ABB RobotStudio station: ESTACION_DEF_ROBOT.rsstn

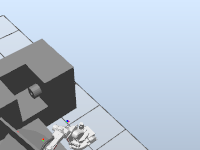
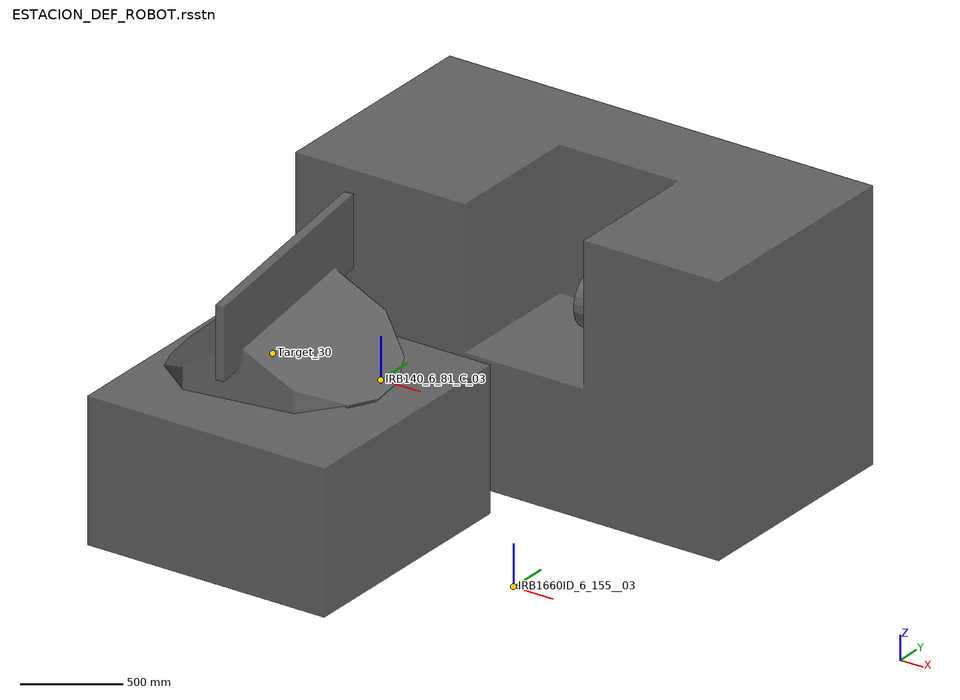
[picture v1: parts stored in the station drawn from their meshes, with robot base, taught points and paths (robot models come from the ABB library and are not in the file)]
Station ESTACION_DEF_ROBOT (saved by RobotStudio 21.2.9526.0)
Controller Controlador6, task T_ROB1: task frame (RAPID world) sits at (1882.6, -1569.1, 39.06) mm, rotated rx 0 ry 0 rz 180 deg in the station
Controller Controlador5
  mechanical unit ROB_1: IRB140_6_81_C_03, 6 joints, base frame (0, 0, 0) mm
Controller Controlador6
  mechanical unit ROB_1: IRB1660ID_6_155__03, 6 joints, base frame (0, 0, 0) mm
Layout (positions relative to the parent item):
  - IRB140_6_81_C_03 [mechanism, from Robots\IRB140_6_81_C_G_03.rslib] at (0, 0, 0) mm; joint values [0, -0.1562, 0.2279, 0, 0.4519, 0] (rad or m)
  - Conjunto_para_piezas_2 [part] at (0, 0, 452.24) mm, rotated rx 90 ry 0 rz 0 deg, size 1400 x 1500 x 1400 mm
  - IRB1660ID_6_155__03 [mechanism, from Robots\IRB1660ID_6_155__03.rslib] at (1882.6, -1569.1, 39.06) mm, rotated rx 0 ry 0 rz 180 deg; joint values [0, 0, 0, 0, 0.5236, 0] (rad or m)
  - Torno [part] at (2480.52, 608.66, 1496.19) mm, rotated rx 0 ry 0 rz 180 deg, size 2500 x 1300 x 1500 mm
  - MyTool_2 [mechanism, from Training Objects\myTool.rslib] at (726.72, -1949.96, 1124.78) mm, rotated rx 180 ry 0 rz 0 deg
Attachment: MyTool_2 is attached to IRB1660ID_6_155__03 / Link6
Targets, tools, work objects and paths stored in the station, written as RAPID:
! task T_ROB1
MODULE Module1
  CONST robtarget Target_10:=[[1714.021,-1416.247,797.687],[1,0,0,0],[0,0,0,0],[9E+09,9E+09,9E+09,9E+09,9E+09,9E+09]];
  CONST robtarget Target_20:=[[1032.438,-2146.001,797.481],[1,0,0,0],[0,0,0,0],[9E+09,9E+09,9E+09,9E+09,9E+09,9E+09]];
  CONST robtarget Target_30:=[[72.148572191,409.131324329,218.503297025],[0.064631034,0.771722064,-0.572722722,0.268805821],[0,0,0,0],[9E+09,9E+09,9E+09,9E+09,9E+09,9E+09]];
  CONST robtarget Target_40:=[[547.54574713,265.221443452,268.080611211],[0.064631034,0.771722064,-0.572722722,0.268805821],[0,0,0,0],[9E+09,9E+09,9E+09,9E+09,9E+09,9E+09]];
  CONST robtarget Target_50:=[[758.013820039,777.48522832,323.070090527],[0.064631034,0.771722064,-0.572722722,0.268805821],[0,0,0,0],[9E+09,9E+09,9E+09,9E+09,9E+09,9E+09]];
  PROC Path_10()
    MoveJ Target_30,v600,z100,tool0\WObj:=Workobject_1;
  ENDPROC
ENDMODULE

! task T_ROB1
MODULE CalibData
  TASK PERS wobjdata Workobject_1:=[FALSE,TRUE,"",[[1255.587,-2234.787,797.481],[0.668146629,0.005699142,0.256021877,0.698570255]],[[65.886,282.487,-93.433],[0.984899065,0.079935059,-0.059861318,-0.141424327]]];
ENDMODULE

! task T_ROB1
MODULE CalibData
  PERS tooldata MyTool:=[TRUE,[[31.792631019,0,229.638935148],[0.945518576,0,0.325568154,0]],[1,[0,0,1],[1,0,0,0],0,0,0]];
  TASK PERS wobjdata Workobject_1:=[FALSE,TRUE,"",[[627.012044235,665.683508341,758.419513401],[0.698570255,0.256021877,-0.005699142,-0.668146629]],[[65.886,282.487,-93.433],[0.984899065,0.079935059,-0.059861318,-0.141424327]]];
ENDMODULE

! task T_ROB1
MODULE Module1
  CONST robtarget Target_30:=[[72.148572191,409.131324329,218.503297025],[0.064631034,0.771722064,-0.572722722,0.268805821],[0,0,0,0],[9E+09,9E+09,9E+09,9E+09,9E+09,9E+09]];
  CONST robtarget Target_40:=[[547.54574713,265.221443452,268.080611211],[0.064631034,0.771722064,-0.572722722,0.268805821],[0,0,0,0],[9E+09,9E+09,9E+09,9E+09,9E+09,9E+09]];
  CONST robtarget Target_50:=[[758.013820039,777.48522832,323.070090527],[0.064631034,0.771722064,-0.572722722,0.268805821],[0,0,0,0],[9E+09,9E+09,9E+09,9E+09,9E+09,9E+09]];
  CONST robtarget Target_30_2:=[[72.148572191,409.131324329,218.503297025],[0.064631034,0.771722064,-0.572722722,0.268805821],[0,0,0,0],[9E+09,9E+09,9E+09,9E+09,9E+09,9E+09]];
  PROC Path_10()
    MoveJ Target_30_2,v600,z100,tool0\WObj:=Workobject_1;
  ENDPROC
ENDMODULE

